// TIA Portal V20 export
DATA_BLOCK "GD_Data"   // DB11
{ S7_Optimized_Access := 'FALSE' }
   VAR RETAIN
      iocontrols : "UDT_Flowmeter_Steuern";
      CurrentValue { S7_SetPoint := 'True'} : DInt;
      zeit_ : Time;
      cycle_1s : Bool;
      count : Int;
      zeit : "UDT_RunTime_Status";
      settime { S7_SetPoint := 'True'} : "UDT_RunTime_Steuern";
      _Sec { S7_SetPoint := 'True'} : Int;
      _Min : Int;
      _Hours : Real;
      first_scan : Bool;
      startup_OK : Bool;
      Reset_Counter : Int;
      Date_Time_is_Lost : Bool;
      Counter_00 : DInt;
      Counter_01 : DInt;
      Testflowsensor_Status : "UDT_Flowmeter_Status";
      Testflowsensor_Control { S7_SetPoint := 'True'} : "UDT_Flowmeter_Steuern";
      Testfuelsensor_Stoe { S7_SetPoint := 'True'} : "UDT_Flowmeter_Stoe";
   END_VAR
BEGIN
END_DATA_BLOCK
